ABB RobotStudio station: gen_alg_jovana.rspag

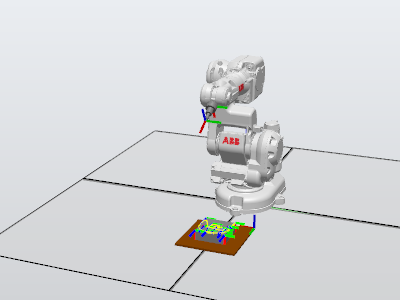
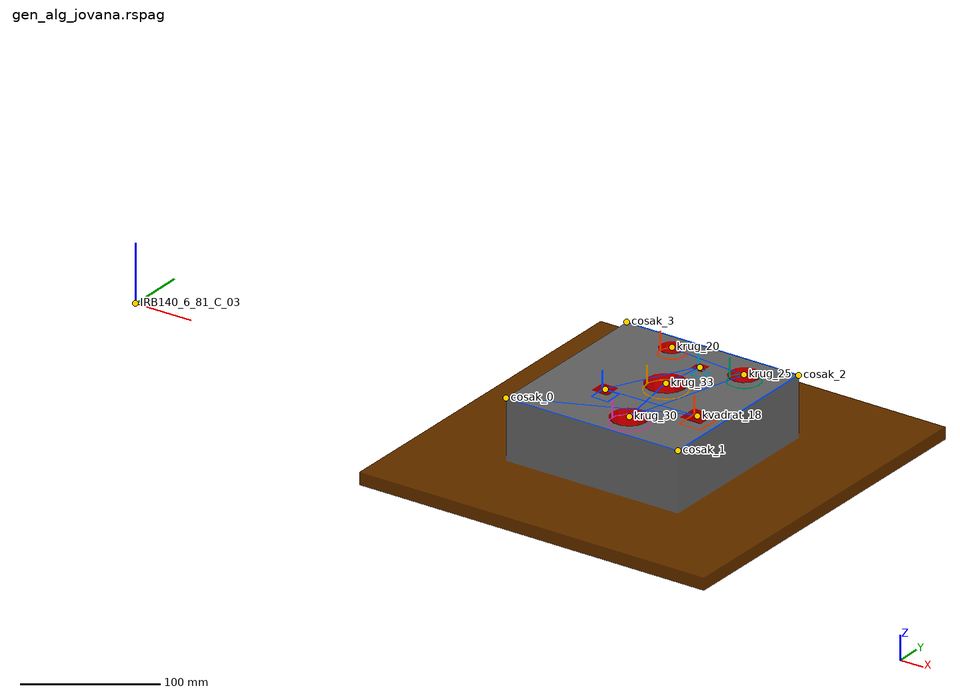
[picture v1: parts stored in the station drawn from their meshes, with robot base, taught points and paths (robot models come from the ABB library and are not in the file)]
--- station ---
Station gen_alg_jovana (saved by RobotStudio 22.3.10190.2)
Controller Controller4
  mechanical unit ROB_1: IRB140_6_81_C_03, 6 joints, base frame (0, 0, 0) mm
Layout (positions relative to the parent item):
  - IRB140_6_81_C_03 [mechanism, from Robots\IRB140_6_81_C_G_03.rslib] at (0, 0, 0) mm; joint values [0, 0, 0, 0, 0.5236, 0] (rad or m)
  - MyGlodalo [mechanism] at (506.29, 0, 679.5) mm, rotated rx 180 ry 60 rz 180 deg
      TCP MyGlodalo at (0, 0, 93) mm, rotated rx 0 ry -90 rz 0 deg
      links: Part_7
  - podloga [part] at (300, 0, 0) mm, size 300 x 300 x 10 mm
  - predmet [part] at (375, 0, 0) mm, size 150 x 150 x 50 mm
Attachment: MyGlodalo is attached to IRB140_6_81_C_03 / Link6
Attachment: wobj_radna_povrsina is attached to podloga

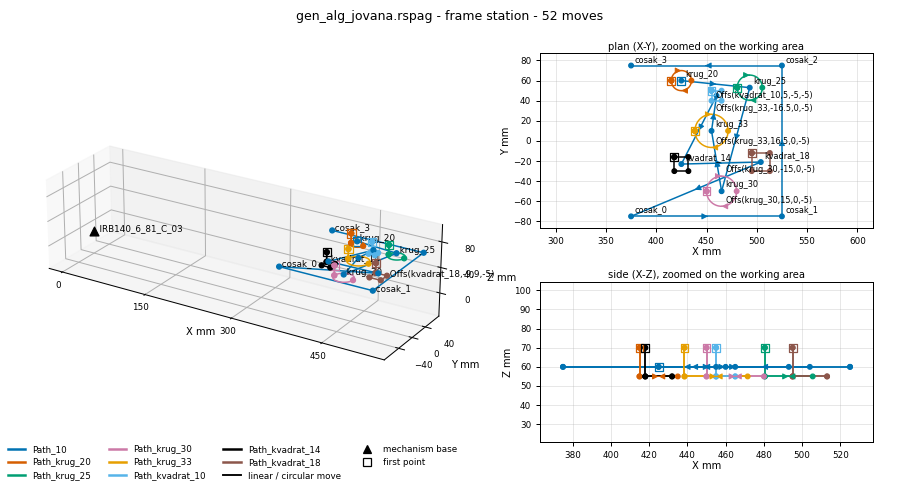
[picture p0: tool path of gen_alg_jovana.rspag in frame station, 52 of 61 moves have a stored position in this frame; points joined in program order, loops and branches not executed]
--- Backups/Controller4/RAPID/TASK1/PROGMOD/CalibData.mod ---
MODULE CalibData
    PERS tooldata MyGlodalo:=[TRUE,[[0,0,93],[0.707106781,0,-0.707106781,0]],[0.3,[0,0,23.122],[1,0,0,0],0,0,0]];
    PERS wobjdata wobj_radna_povrsina:=[FALSE,TRUE,"",[[300,150,10],[0.707106781,0,0,-0.707106781]],[[0,0,0],[1,0,0,0]]];
ENDMODULE

--- Backups/Controller4/RAPID/TASK1/PROGMOD/Module1.mod ---
MODULE Module1
        CONST robtarget krug_20:=[[90,125,50],[0.5,-0.5,0.5,0.5],[0,0,0,0],[9E+09,9E+09,9E+09,9E+09,9E+09,9E+09]];
    CONST robtarget krug_25:=[[97,193,50],[0.5,-0.5,0.5,0.5],[0,0,0,0],[9E+09,9E+09,9E+09,9E+09,9E+09,9E+09]];
    CONST robtarget krug_30:=[[200,165,50],[0.5,-0.5,0.5,0.5],[-1,0,-1,0],[9E+09,9E+09,9E+09,9E+09,9E+09,9E+09]];
    CONST robtarget krug_33:=[[140,155,50],[0.5,-0.5,0.5,0.5],[0,0,0,0],[9E+09,9E+09,9E+09,9E+09,9E+09,9E+09]];
    CONST robtarget kvadrat_10:=[[105,160,50],[0.5,-0.5,0.5,0.5],[0,0,0,0],[9E+09,9E+09,9E+09,9E+09,9E+09,9E+09]];
    CONST robtarget kvadrat_14:=[[173,125,50],[0.5,-0.5,0.5,0.5],[0,0,0,0],[9E+09,9E+09,9E+09,9E+09,9E+09,9E+09]];
    CONST robtarget kvadrat_18:=[[171,204,50],[0.5,-0.5,0.5,0.5],[0,0,0,0],[9E+09,9E+09,9E+09,9E+09,9E+09,9E+09]];
    CONST robtarget cosak_0:=[[225,75,50],[0.5,-0.5,0.5,0.5],[-1,0,-1,0],[9E+09,9E+09,9E+09,9E+09,9E+09,9E+09]];
    CONST robtarget cosak_1:=[[225,225,50],[0.5,-0.5,0.5,0.5],[0,0,0,0],[9E+09,9E+09,9E+09,9E+09,9E+09,9E+09]];
    CONST robtarget cosak_2:=[[75,225,50],[0.5,-0.5,0.5,0.5],[0,0,0,0],[9E+09,9E+09,9E+09,9E+09,9E+09,9E+09]];
    CONST robtarget cosak_3:=[[75,75,50],[0.5,-0.5,0.5,0.5],[0,0,0,0],[9E+09,9E+09,9E+09,9E+09,9E+09,9E+09]];
!***********************************************************
    !
    ! Module:  Module1
    !
    ! Description:
    !   <Insert description here>
    !
    ! Author: Studen
    !
    ! Version: 1.0
    !
    !***********************************************************


    !***********************************************************
    !
    ! Procedure main
    !
    !   This is the entry point of your program
    !
    !***********************************************************
    PROC Path_10()
        MoveL krug_20,v1000,z100,MyGlodalo\WObj:=wobj_radna_povrsina;
        MoveL krug_25,v1000,z100,MyGlodalo\WObj:=wobj_radna_povrsina;
        MoveL krug_30,v1000,z100,MyGlodalo\WObj:=wobj_radna_povrsina;
        MoveL krug_33,v1000,z100,MyGlodalo\WObj:=wobj_radna_povrsina;
        MoveL kvadrat_10,v1000,z100,MyGlodalo\WObj:=wobj_radna_povrsina;
        MoveL kvadrat_14,v1000,z100,MyGlodalo\WObj:=wobj_radna_povrsina;
        MoveL kvadrat_18,v1000,z100,MyGlodalo\WObj:=wobj_radna_povrsina;
        MoveL cosak_0,v1000,z100,MyGlodalo\WObj:=wobj_radna_povrsina;
        MoveL cosak_1,v1000,z100,MyGlodalo\WObj:=wobj_radna_povrsina;
        MoveL cosak_2,v1000,z100,MyGlodalo\WObj:=wobj_radna_povrsina;
        MoveL cosak_3,v1000,z100,MyGlodalo\WObj:=wobj_radna_povrsina;
    ENDPROC

    PROC Path_krug_20()
        MoveL Offs(krug_20, 0, -10, 10),currentSpeed,z0,MyGlodalo\WObj:=wobj_radna_povrsina;
        MoveL Offs(krug_20, 0, -10, -5),currentSpeed,z0,MyGlodalo\WObj:=wobj_radna_povrsina;
        MoveC Offs(krug_20, -10, 0, -5), Offs(krug_20, 0, 10, -5),currentSpeed,z0,MyGlodalo\WObj:=wobj_radna_povrsina;
        MoveC Offs(krug_20, 10, 0, -5), Offs(krug_20, 0, -10, -5),currentSpeed,z0,MyGlodalo\WObj:=wobj_radna_povrsina;
        MoveL Offs(krug_20, 0, -10, 10),currentSpeed,z0,MyGlodalo\WObj:=wobj_radna_povrsina;
    ENDPROC
    PROC Path_krug_25()
        MoveL Offs(krug_25, 0, -12.5, 10),currentSpeed,z0,MyGlodalo\WObj:=wobj_radna_povrsina;
        MoveL Offs(krug_25, 0, -12.5, -5),currentSpeed,z0,MyGlodalo\WObj:=wobj_radna_povrsina;
        MoveC Offs(krug_25, -12.5, 0, -5), Offs(krug_25, 0, 12.5, -5),currentSpeed,z0,MyGlodalo\WObj:=wobj_radna_povrsina;
        MoveC Offs(krug_25, 12.5, 0, -5), Offs(krug_25, 0, -12.5, -5),currentSpeed,z0,MyGlodalo\WObj:=wobj_radna_povrsina;
        MoveL Offs(krug_25, 0, -12.5, 10),currentSpeed,z0,MyGlodalo\WObj:=wobj_radna_povrsina;
    ENDPROC
    PROC Path_krug_30()
        MoveL Offs(krug_30, 0, -15, 10),currentSpeed,z0,MyGlodalo\WObj:=wobj_radna_povrsina;
        MoveL Offs(krug_30, 0, -15, -5),currentSpeed,z0,MyGlodalo\WObj:=wobj_radna_povrsina;
        MoveC Offs(krug_30, -15, 0, -5), Offs(krug_30, 0, 15, -5),currentSpeed,z0,MyGlodalo\WObj:=wobj_radna_povrsina;
        MoveC Offs(krug_30, 15, 0, -5), Offs(krug_30, 0, -15, -5),currentSpeed,z0,MyGlodalo\WObj:=wobj_radna_povrsina;
        MoveL Offs(krug_30, 0, -15, 10),currentSpeed,z0,MyGlodalo\WObj:=wobj_radna_povrsina;
    ENDPROC
    PROC Path_krug_33()
        MoveL Offs(krug_33, 0, -16.5, 10),currentSpeed,z0,MyGlodalo\WObj:=wobj_radna_povrsina;
        MoveL Offs(krug_33, 0, -16.5, -5),currentSpeed,z0,MyGlodalo\WObj:=wobj_radna_povrsina;
        MoveC Offs(krug_33, -16.5, 0, -5), Offs(krug_33, 0, 16.5, -5),currentSpeed,z0,MyGlodalo\WObj:=wobj_radna_povrsina;
        MoveC Offs(krug_33, 16.5, 0, -5), Offs(krug_33, 0, -16.5, -5),currentSpeed,z0,MyGlodalo\WObj:=wobj_radna_povrsina;
        MoveL Offs(krug_33, 0, -16.5, 10),currentSpeed,z0,MyGlodalo\WObj:=wobj_radna_povrsina;
    ENDPROC
    PROC Path_kvadrat_10()
        MoveL Offs(kvadrat_10, -5, -5, 10),currentSpeed,z0,MyGlodalo\WObj:=wobj_radna_povrsina;
        MoveL Offs(kvadrat_10, -5, -5, -5),currentSpeed,z0,MyGlodalo\WObj:=wobj_radna_povrsina;
        MoveL Offs(kvadrat_10, 5, -5, -5),currentSpeed,z0,MyGlodalo\WObj:=wobj_radna_povrsina;
        MoveL Offs(kvadrat_10, 5, 5, -5),currentSpeed,z0,MyGlodalo\WObj:=wobj_radna_povrsina;
        MoveL Offs(kvadrat_10, -5, 5, -5),currentSpeed,z0,MyGlodalo\WObj:=wobj_radna_povrsina;
        MoveL Offs(kvadrat_10, -5, -5, -5),currentSpeed,z0,MyGlodalo\WObj:=wobj_radna_povrsina;
        MoveL Offs(kvadrat_10, -5, -5, 10),currentSpeed,z0,MyGlodalo\WObj:=wobj_radna_povrsina;
    ENDPROC
    PROC Path_kvadrat_14()
        MoveL Offs(kvadrat_14, -7, -7, 10),currentSpeed,z0,MyGlodalo\WObj:=wobj_radna_povrsina;
        MoveL Offs(kvadrat_14, -7, -7, -5),currentSpeed,z0,MyGlodalo\WObj:=wobj_radna_povrsina;
        MoveL Offs(kvadrat_14, 7, -7, -5),currentSpeed,z0,MyGlodalo\WObj:=wobj_radna_povrsina;
        MoveL Offs(kvadrat_14, 7, 7, -5),currentSpeed,z0,MyGlodalo\WObj:=wobj_radna_povrsina;
        MoveL Offs(kvadrat_14, -7, 7, -5),currentSpeed,z0,MyGlodalo\WObj:=wobj_radna_povrsina;
        MoveL Offs(kvadrat_14, -7, -7, -5),currentSpeed,z0,MyGlodalo\WObj:=wobj_radna_povrsina;
        MoveL Offs(kvadrat_14, -7, -7, 10),currentSpeed,z0,MyGlodalo\WObj:=wobj_radna_povrsina;
    ENDPROC
    PROC Path_kvadrat_18()
        MoveL Offs(kvadrat_18, -9, -9, 10),currentSpeed,z0,MyGlodalo\WObj:=wobj_radna_povrsina;
        MoveL Offs(kvadrat_18, -9, -9, -5),currentSpeed,z0,MyGlodalo\WObj:=wobj_radna_povrsina;
        MoveL Offs(kvadrat_18, 9, -9, -5),currentSpeed,z0,MyGlodalo\WObj:=wobj_radna_povrsina;
        MoveL Offs(kvadrat_18, 9, 9, -5),currentSpeed,z0,MyGlodalo\WObj:=wobj_radna_povrsina;
        MoveL Offs(kvadrat_18, -9, 9, -5),currentSpeed,z0,MyGlodalo\WObj:=wobj_radna_povrsina;
        MoveL Offs(kvadrat_18, -9, -9, -5),currentSpeed,z0,MyGlodalo\WObj:=wobj_radna_povrsina;
        MoveL Offs(kvadrat_18, -9, -9, 10),currentSpeed,z0,MyGlodalo\WObj:=wobj_radna_povrsina;
    ENDPROC
    PROC Path_stranica(bool direction, num stranica)
        VAR robtarget start_target;
        VAR robtarget end_target;
        VAR robtarget temp_target;
        TEST stranica
            CASE 0:
                start_target := cosak_0;
                end_target := cosak_1;
            CASE 1:
                start_target := cosak_1;
                end_target := cosak_2;
            CASE 2:
                start_target := cosak_2;
                end_target := cosak_3;
            CASE 3:
                start_target := cosak_3;
                end_target := cosak_0;
        ENDTEST

        IF not direction THEN
            temp_target := start_target;
            start_target := end_target;
            end_target := temp_target;
        ENDIF
        MoveL Offs(start_target, 0, 0, 10),currentSpeed,z0,MyGlodalo\WObj:=wobj_radna_povrsina;
        MoveL Offs(start_target, 0, 0, -5),currentSpeed,z0,MyGlodalo\WObj:=wobj_radna_povrsina;
        MoveL Offs(end_target, 0, 0, -5),currentSpeed,z0,MyGlodalo\WObj:=wobj_radna_povrsina;
        MoveL Offs(end_target, 0, 0, 10),currentSpeed,z0,MyGlodalo\WObj:=wobj_radna_povrsina;
    ENDPROC
ENDMODULE

--- Backups/Controller4/RAPID/TASK1/PROGMOD/SERVER.mod ---
MODULE SERVER

    !////////////////
    !GLOBAL VARIABLES
    !////////////////

    !//Robot configuration
    PERS tooldata currentTool:=[TRUE,[[0,0,0],[1,0,0,0]],[0.001,[0,0,0.001],[1,0,0,0],0,0,0]];
    PERS wobjdata currentWobj:=[FALSE,TRUE,"",[[0,0,0],[1,0,0,0]],[[0,0,0],[1,0,0,0]]];
    PERS speeddata currentSpeed;
    PERS zonedata currentZone;

    !// Clock Synchronization
    PERS bool startLog:=TRUE;
    PERS bool startRob:=TRUE;

    !// Mutex between logger and changing the tool and work objects
    PERS bool frameMutex:=FALSE;

    !//PC communication
    VAR socketdev clientSocket;
    VAR socketdev serverSocket;
    VAR num instructionCode;
    VAR num params{10};
    VAR num nParams;

    !PERS string ipController:= "192.168.125.1"; !robot default IP
    PERS string ipController:="127.0.0.1";
    !local IP for testing in simulation
    PERS num serverPort:=5000;

    !//Motion of the robot
    VAR robtarget cartesianTarget;
    VAR jointtarget jointsTarget;
    VAR bool moveCompleted;
    !Set to true after finishing a Move instruction.

    !//Buffered move variables
    CONST num MAX_BUFFER:=512;
    VAR num BUFFER_POS:=0;
    VAR robtarget bufferTargets{MAX_BUFFER};
    VAR speeddata bufferSpeeds{MAX_BUFFER};

    !//External axis position variables
    VAR extjoint externalAxis;

    !//Circular move buffer
    VAR robtarget circPoint;

    !//Correct Instruction Execution and possible return values
    VAR num ok;
    CONST num SERVER_BAD_MSG:=0;
    CONST num SERVER_OK:=1;


    !////////////////
    !LOCAL METHODS
    !////////////////

    !//Method to parse the message received from a PC
    !// If correct message, loads values on:
    !// - instructionCode.
    !// - nParams: Number of received parameters.
    !// - params{nParams}: Vector of received params.
    PROC ParseMsg(string msg)
        !//Local variables
        VAR bool auxOk;
        VAR num ind:=1;
        VAR num newInd;
        VAR num length;
        VAR num indParam:=1;
        VAR string subString;
        VAR bool end:=FALSE;

        !//Find the end character
        length:=StrMatch(msg,1,"#");
        IF length>StrLen(msg) THEN
            !//Corrupt message
            nParams:=-1;
        ELSE
            !//Read Instruction code
            newInd:=StrMatch(msg,ind," ")+1;
            subString:=StrPart(msg,ind,newInd-ind-1);
            auxOk:=StrToVal(subString,instructionCode);
            IF auxOk=FALSE THEN
                !//Impossible to read instruction code
                nParams:=-1;
            ELSE
                ind:=newInd;
                !//Read all instruction parameters (maximum of 8)
                WHILE end=FALSE DO
                    newInd:=StrMatch(msg,ind," ")+1;
                    IF newInd>length THEN
                        end:=TRUE;
                    ELSE
                        subString:=StrPart(msg,ind,newInd-ind-1);
                        auxOk:=StrToVal(subString,params{indParam});
                        indParam:=indParam+1;
                        ind:=newInd;
                    ENDIF
                ENDWHILE
                nParams:=indParam-1;
            ENDIF
        ENDIF
    ENDPROC


    !//Handshake between server and client:
    !// - Creates socket.
    !// - Waits for incoming TCP connection.
    PROC ServerCreateAndConnect(string ip,num port)
        VAR string clientIP;

        SocketCreate serverSocket;
        SocketBind serverSocket,ip,port;
        SocketListen serverSocket;
        TPWrite "SERVER: Server waiting for incoming connections ...";
        WHILE SocketGetStatus(clientSocket)<>SOCKET_CONNECTED DO
            SocketAccept serverSocket,clientSocket\ClientAddress:=clientIP\Time:=WAIT_MAX;
            IF SocketGetStatus(clientSocket)<>SOCKET_CONNECTED THEN
                TPWrite "SERVER: Problem serving an incoming connection.";
                TPWrite "SERVER: Try reconnecting.";
            ENDIF
            !//Wait 0.5 seconds for the next reconnection
            WaitTime 0.5;
        ENDWHILE
        TPWrite "SERVER: Connected to IP "+clientIP;
    ENDPROC


    !//Parameter initialization
    !// Loads default values for
    !// - Tool.
    !// - WorkObject.
    !// - Zone.
    !// - Speed.
    PROC Initialize()
        currentTool:=[TRUE,[[0,0,0],[1,0,0,0]],[0.001,[0,0,0.001],[1,0,0,0],0,0,0]];
        currentWobj:=[FALSE,TRUE,"",[[0,0,0],[1,0,0,0]],[[0,0,0],[1,0,0,0]]];
        currentSpeed:=[100,50,0,0];
        currentZone:=[FALSE,0.3,0.3,0.3,0.03,0.3,0.03];
        !z0

        !Find the current external axis values so they don't move when we start
        jointsTarget:=CJointT();
        externalAxis:=jointsTarget.extax;
    ENDPROC


    !////////////////////////
    !//SERVER: Main procedure
    !////////////////////////
    PROC main()
        !//Local variables
        VAR string receivedString;
        !//Received string
        VAR string sendString;
        !//Reply string
        VAR string addString;
        !//String to add to the reply.
        VAR bool connected;
        !//Client connected
        VAR bool reconnected;
        !//Drop and reconnection happened during serving a command
        VAR robtarget cartesianPose;
        VAR jointtarget jointsPose;
!        Path_10;
        !//Motion configuration
        ConfL\Off;
        SingArea\Wrist;
        moveCompleted:=TRUE;

        !//Initialization of WorkObject, Tool, Speed and Zone
        Initialize;

        !//Socket connection
        connected:=FALSE;
        ServerCreateAndConnect ipController,serverPort;
        connected:=TRUE;

        !//Server Loop
        WHILE TRUE DO
            !//Initialization of program flow variables
            ok:=SERVER_OK;
            !//Correctness of executed instruction.
            reconnected:=FALSE;
            !//Has communication dropped after receiving a command?
            addString:="";

            !//Wait for a command
            SocketReceive clientSocket\Str:=receivedString\Time:=WAIT_MAX;
            ParseMsg receivedString;

            !//Execution of the command
            TEST instructionCode
            CASE 0:
                !Ping
                IF nParams=0 THEN
                    ok:=SERVER_OK;
                ELSE
                    ok:=SERVER_BAD_MSG;
                ENDIF

            CASE 1:
                !Cartesian Move
                IF nParams=7 THEN
                    cartesianTarget:=[[params{1},params{2},params{3}],
                                       [params{4},params{5},params{6},params{7}],
                                       [0,0,0,0],
                                       externalAxis];
                    ok:=SERVER_OK;
                    moveCompleted:=FALSE;
                    MoveL cartesianTarget,currentSpeed,currentZone,currentTool\WObj:=currentWobj;
                    moveCompleted:=TRUE;
                ELSE
                    ok:=SERVER_BAD_MSG;
                ENDIF

            CASE 2:
                !Joint Move
                IF nParams=6 THEN
                    jointsTarget:=[[params{1},params{2},params{3},params{4},params{5},params{6}],externalAxis];
                    ok:=SERVER_OK;
                    moveCompleted:=FALSE;
                    MoveAbsJ jointsTarget,currentSpeed,currentZone,currentTool\Wobj:=currentWobj;
                    moveCompleted:=TRUE;
                ELSE
                    ok:=SERVER_BAD_MSG;
                ENDIF

            CASE 3:
                !Get Cartesian Coordinates (with current tool and workobject)
                IF nParams=0 THEN
                    cartesianPose:=CRobT(\Tool:=currentTool\WObj:=currentWObj);
                    addString:=NumToStr(cartesianPose.trans.x,2)+" ";
                    addString:=addString+NumToStr(cartesianPose.trans.y,2)+" ";
                    addString:=addString+NumToStr(cartesianPose.trans.z,2)+" ";
                    addString:=addString+NumToStr(cartesianPose.rot.q1,3)+" ";
                    addString:=addString+NumToStr(cartesianPose.rot.q2,3)+" ";
                    addString:=addString+NumToStr(cartesianPose.rot.q3,3)+" ";
                    addString:=addString+NumToStr(cartesianPose.rot.q4,3);
                    !End of string
                    ok:=SERVER_OK;
                ELSE
                    ok:=SERVER_BAD_MSG;
                ENDIF

            CASE 4:
                !Get Joint Coordinates
                IF nParams=0 THEN
                    jointsPose:=CJointT();
                    addString:=NumToStr(jointsPose.robax.rax_1,2)+" ";
                    addString:=addString+NumToStr(jointsPose.robax.rax_2,2)+" ";
                    addString:=addString+NumToStr(jointsPose.robax.rax_3,2)+" ";
                    addString:=addString+NumToStr(jointsPose.robax.rax_4,2)+" ";
                    addString:=addString+NumToStr(jointsPose.robax.rax_5,2)+" ";
                    addString:=addString+NumToStr(jointsPose.robax.rax_6,2);
                    !End of string
                    ok:=SERVER_OK;
                ELSE
                    ok:=SERVER_BAD_MSG;
                ENDIF
            CASE 5:
                !Get external axis positions
                IF nParams=0 THEN
                    jointsPose:=CJointT();
                    addString:=StrPart(NumToStr(jointsTarget.extax.eax_a,2),1,8)+" ";
                    addString:=addString+StrPart(NumToStr(jointsTarget.extax.eax_b,2),1,8)+" ";
                    addString:=addString+StrPart(NumToStr(jointsTarget.extax.eax_c,2),1,8)+" ";
                    addString:=addString+StrPart(NumToStr(jointsTarget.extax.eax_d,2),1,8)+" ";
                    addString:=addString+StrPart(NumToStr(jointsTarget.extax.eax_e,2),1,8)+" ";
                    addString:=addString+StrPart(NumToStr(jointsTarget.extax.eax_f,2),1,8);
                    !End of string
                    ok:=SERVER_OK;
                ELSE
                    ok:=SERVER_BAD_MSG;
                ENDIF

            CASE 6:
                !Set Tool
                IF nParams=7 THEN
                    WHILE (frameMutex) DO
                        WaitTime .01;
                        !// If the frame is being used by logger, wait here
                    ENDWHILE
                    frameMutex:=TRUE;
                    currentTool.tframe.trans.x:=params{1};
                    currentTool.tframe.trans.y:=params{2};
                    currentTool.tframe.trans.z:=params{3};
                    currentTool.tframe.rot.q1:=params{4};
                    currentTool.tframe.rot.q2:=params{5};
                    currentTool.tframe.rot.q3:=params{6};
                    currentTool.tframe.rot.q4:=params{7};
                    ok:=SERVER_OK;
                    frameMutex:=FALSE;
                ELSE
                    ok:=SERVER_BAD_MSG;
                ENDIF

            CASE 7:
                !Set Work Object
                IF nParams=7 THEN
                    currentWobj.oframe.trans.x:=params{1};
                    currentWobj.oframe.trans.y:=params{2};
                    currentWobj.oframe.trans.z:=params{3};
                    currentWobj.oframe.rot.q1:=params{4};
                    currentWobj.oframe.rot.q2:=params{5};
                    currentWobj.oframe.rot.q3:=params{6};
                    currentWobj.oframe.rot.q4:=params{7};
                    ok:=SERVER_OK;
                ELSE
                    ok:=SERVER_BAD_MSG;
                ENDIF

            CASE 8:
                !Set Speed of the Robot
                IF nParams=4 THEN
                    currentSpeed.v_tcp:=params{1};
                    currentSpeed.v_ori:=params{2};
                    currentSpeed.v_leax:=params{3};
                    currentSpeed.v_reax:=params{4};
                    ok:=SERVER_OK;
                ELSEIF nParams=2 THEN
                    currentSpeed.v_tcp:=params{1};
                    currentSpeed.v_ori:=params{2};
                    ok:=SERVER_OK;
                ELSE
                    ok:=SERVER_BAD_MSG;
                ENDIF

            CASE 9:
                !Set zone data
                IF nParams=4 THEN
                    IF params{1}=1 THEN
                        currentZone.finep:=TRUE;
                        currentZone.pzone_tcp:=0.0;
                        currentZone.pzone_ori:=0.0;
                        currentZone.zone_ori:=0.0;
                    ELSE
                        currentZone.finep:=FALSE;
                        currentZone.pzone_tcp:=params{2};
                        currentZone.pzone_ori:=params{3};
                        currentZone.zone_ori:=params{4};
                    ENDIF
                    ok:=SERVER_OK;
                ELSE
                    ok:=SERVER_BAD_MSG;
                ENDIF

            CASE 30:
                !Add Cartesian Coordinates to buffer
                IF nParams=7 THEN
                    cartesianTarget:=[[params{1},params{2},params{3}],
                                        [params{4},params{5},params{6},params{7}],
                                        [0,0,0,0],
                                        externalAxis];
                    IF BUFFER_POS<MAX_BUFFER THEN
                        BUFFER_POS:=BUFFER_POS+1;
                        bufferTargets{BUFFER_POS}:=cartesianTarget;
                        bufferSpeeds{BUFFER_POS}:=currentSpeed;
                    ENDIF
                    ok:=SERVER_OK;
                ELSE
                    ok:=SERVER_BAD_MSG;
                ENDIF

            CASE 31:
                !Clear Cartesian Buffer
                IF nParams=0 THEN
                    BUFFER_POS:=0;
                    ok:=SERVER_OK;
                ELSE
                    ok:=SERVER_BAD_MSG;
                ENDIF

            CASE 32:
                !Get Buffer Size)
                IF nParams=0 THEN
                    addString:=NumToStr(BUFFER_POS,2);
                    ok:=SERVER_OK;
                ELSE
                    ok:=SERVER_BAD_MSG;
                ENDIF

            CASE 33:
                !Execute moves in cartesianBuffer as linear moves
                IF nParams=0 THEN
                    FOR i FROM 1 TO (BUFFER_POS) DO
                        MoveL bufferTargets{i},bufferSpeeds{i},currentZone,currentTool\WObj:=currentWobj;
                    ENDFOR
                    ok:=SERVER_OK;
                ELSE
                    ok:=SERVER_BAD_MSG;
                ENDIF

            CASE 34:
                !External Axis move
                IF nParams=6 THEN
                    externalAxis:=[params{1},params{2},params{3},params{4},params{5},params{6}];
                    jointsTarget:=CJointT();
                    jointsTarget.extax:=externalAxis;
                    ok:=SERVER_OK;
                    moveCompleted:=FALSE;
                    MoveAbsJ jointsTarget,currentSpeed,currentZone,currentTool\Wobj:=currentWobj;
                    moveCompleted:=TRUE;
                ELSE
                    ok:=SERVER_BAD_MSG;
                ENDIF

            CASE 35:
                !Specify circPoint for circular move, and then wait on toPoint
                IF nParams=7 THEN
                    circPoint:=[[params{1},params{2},params{3}],
                                [params{4},params{5},params{6},params{7}],
                                [0,0,0,0],
                                externalAxis];
                    ok:=SERVER_OK;
                ELSE
                    ok:=SERVER_BAD_MSG;
                ENDIF

            CASE 36:
                !specify toPoint, and use circPoint specified previously
                IF nParams=7 THEN
                    cartesianTarget:=[[params{1},params{2},params{3}],
                                        [params{4},params{5},params{6},params{7}],
                                        [0,0,0,0],
                                        externalAxis];
                    MoveC circPoint,cartesianTarget,currentSpeed,currentZone,currentTool\WObj:=currentWobj;
                    ok:=SERVER_OK;
                ELSE
                    ok:=SERVER_BAD_MSG;
                ENDIF
            CASE 60:
                ! DO PATH
                IF nParams=2 THEN
                    IF params{2}=0 THEN
                        Path_stranica FALSE, params{1};
                    ELSE
                        Path_stranica TRUE, params{1};
                    ENDIF
                ENDIF
                IF nParams=1 THEN
                    TEST params{1}
                        CASE 10:
                            Path_kvadrat_10;
                        CASE 14:
                            Path_kvadrat_14;
                        CASE 18:
                            Path_kvadrat_18;
                        CASE 20:
                            Path_krug_20;
                        CASE 25:
                            Path_krug_25;
                        CASE 30:
                            Path_krug_30;
                        CASE 33:
                            Path_krug_33;
                    ENDTEST
                ENDIF

            CASE 98:
                !returns current robot info: serial number, robotware version, and robot type
                IF nParams=0 THEN
                    addString:=GetSysInfo(\SerialNo)+"*";
                    addString:=addString+GetSysInfo(\SWVersion)+"*";
                    addString:=addString+GetSysInfo(\RobotType);
                    ok:=SERVER_OK;
                ELSE
                    ok:=SERVER_BAD_MSG;
                ENDIF

            CASE 99:
                !Close Connection
                IF nParams=0 THEN
                    TPWrite "SERVER: Client has closed connection.";
                    connected:=FALSE;
                    !//Closing the server
                    SocketClose clientSocket;
                    SocketClose serverSocket;

                    !Reinitiate the server
                    ServerCreateAndConnect ipController,serverPort;
                    connected:=TRUE;
                    reconnected:=TRUE;
                    ok:=SERVER_OK;
                ELSE
                    ok:=SERVER_BAD_MSG;
                ENDIF
            DEFAULT:
                TPWrite "SERVER: Illegal instruction code";
                ok:=SERVER_BAD_MSG;
            ENDTEST

            !Compose the acknowledge string to send back to the client
            IF connected=TRUE THEN
                IF reconnected=FALSE THEN
                    IF SocketGetStatus(clientSocket)=SOCKET_CONNECTED THEN
                        sendString:=NumToStr(instructionCode,0);
                        sendString:=sendString+" "+NumToStr(ok,0);
                        sendString:=sendString+" "+addString;
                        SocketSend clientSocket\Str:=sendString;
                    ENDIF
                ENDIF
            ENDIF
        ENDWHILE

    ERROR (LONG_JMP_ALL_ERR)
        TPWrite "SERVER: ------";
        TPWrite "SERVER: Error Handler:"+NumtoStr(ERRNO,0);
        TEST ERRNO
        CASE ERR_SOCK_CLOSED:
            TPWrite "SERVER: Lost connection to the client.";
            TPWrite "SERVER: Closing socket and restarting.";
            TPWrite "SERVER: ------";
            connected:=FALSE;
            !//Closing the server
            SocketClose clientSocket;
            SocketClose serverSocket;
            !//Reinitiate the server
            ServerCreateAndConnect ipController,serverPort;
            reconnected:=FALSE;
            connected:=TRUE;
            RETRY;
        DEFAULT:
            TPWrite "SERVER: Unknown error.";
            TPWrite "SERVER: Closing socket and restarting.";
            TPWrite "SERVER: ------";
            connected:=FALSE;
            !//Closing the server
            SocketClose clientSocket;
            SocketClose serverSocket;
            !//Reinitiate the server
            ServerCreateAndConnect ipController,serverPort;
            reconnected:=FALSE;
            connected:=TRUE;
            RETRY;
        ENDTEST
    ENDPROC

ENDMODULE
